PROGRAM MAIN

VAR
END_VAR

END_PROGRAM

(* stored: Version 1.1.0.1, ProductVersion 3.1.4024.12
   POU MAIN: Id {02f712db-0be8-4927-8ccc-74642d8979eb}, SpecialFunc None *)
